(* PLC project static_torsion.project, CODESYS CODESYS V3.5 SP17 Patch 3 *)
(* stored: creationDateTime 1970-01-01T00:00:00, modificationDateTime 2026-06-22T15:12:39.4699931 *)

FUNCTION_BLOCK FB_IntRingBuffer
  VAR_INPUT
    InVal : INT;  (* Новое значение каждый цикл *)
    Reset : BOOL;  (* Сброс буфера *)
  END_VAR
  VAR_OUTPUT
    Out : ARRAY[0..(Size - 1)] OF INT;
    Out_WORDS : ARRAY[0..(Size - 1)] OF WORD;
    BUFFER_SIZE : UINT := Size;
    head : UINT;  (* Индекс следующей записи в [0..Size-1] *)
  END_VAR
  VAR CONSTANT
    Size : UINT := 50;  (* Размер буфера *)
  END_VAR
  VAR
    store : ARRAY[0..(Size - 1)] OF INT;  (* Внутреннее кольцо *)
    filled : BOOL;  (* Окно уже полностью заполнено *)
    i : UINT;
    oldestIdx : UINT;
    idx : UINT;
  END_VAR

            // Обработка сброса
IF Reset THEN
    // Очистка
    FOR i := 0 TO Size - 1 DO
        store[i] := 0;
    END_FOR;
    head := 0;
    filled := FALSE;
END_IF;

// Запись нового значения в кольцо
store[head] := InVal;
head := head + 1;
IF head >= Size THEN
    head := 0;
    filled := TRUE; // как минимум один полный оборот сделан
END_IF;

// Формирование окна Out[1..SizeActual] от старого к новому
IF filled THEN
    oldestIdx := head; // после записи head указывает на "следующий"; он же — самый старый
ELSE
    oldestIdx := 0;    // пока не заполнены, начинаем с 0
END_IF;

FOR i := 0 TO Size - 1 DO
    idx := oldestIdx + i;
    IF idx >= Size THEN
        idx := idx - Size; // быстрый модуль
    END_IF;
    Out[i] := store[idx];
	Out_WORDS[i] := TO_WORD(Out[i]);
END_FOR;
          
END_FUNCTION_BLOCK
